// TwinCAT 3 PLC project plc1
// ProgramVersion: 3.1.4024.0
// libraries:
//   SPT Base Types, * (Beckhoff Automation LLC)
//   SPT_XPlanar, * (Beckhoff Automation LLC)
//   Tc2_Standard, * (Beckhoff Automation GmbH)
//   Tc2_System, * (Beckhoff Automation GmbH)
//   Tc3_Mc3PlanarMotion, * (Beckhoff Automation GmbH)
//   Tc3_Module, * (Beckhoff Automation GmbH)
//   Tc3_Physics, * (Beckhoff Automation GmbH)
//   Tc3_XPlanarStandard, * (Beckhoff Automation GmbH)
//   Tc3_XPlanarUtility, * (Beckhoff Automation GmbH & Co. KG)
//   VisuDialogs, * (System)
// project tree:
//   DUTs/ ST_MoverData.TcDUT, ST_StationData.TcDUT
//   / GlobalTextList.TcGTLO, PlcTask.TcTTO, Visualization Manager.TcVMO (not stored)
//   GVLs/ GVL.TcGVL
//   POUs/ FB_ProcessStation.TcPOU, FB_XPlanarModule.TcPOU, MAIN.TcPOU
//   VISUs/ Visualization.TcVIS
//   VISUs/XPlanarObjects/ VisuLayout.TcVIS, VisuMover.TcVIS, VisuStation.TcVIS
// real-time tasks:
//   TASK PlcTask: cycle T#10ms, priority 20, ADS port 350
//   TASK XPlanar Task16: cycle T#250us, priority 1, ADS port 351
//   TASK XPlanar Task17: cycle T#250us, priority 2, ADS port 352
//   TASK MC-Task (MET): cycle T#2ms, priority 3, ADS port 353
//   TASK MC-Task (MPT): cycle T#10ms, priority 4, ADS port 354
//   TASK Job Task: cycle default, priority 5
// variable links:
//   XPlanar MC Project/Axes/Mover4220_1 <-> TcCOM Objects/XPlanar/Mover4220_1
//     IoToMc/STD <-> OutputsToNC3/HWToNC3
//     McToIo/STD <-> InputsFromNC3/NC3ToHW
//   XPlanar MC Project/Axes/Mover4220_2 <-> TcCOM Objects/XPlanar/Mover4220_2
//     McToIo/STD <-> InputsFromNC3/NC3ToHW
//   XPlanar MC Project/Axes/Mover4220_3 <-> TcCOM Objects/XPlanar/Mover4220_3
//     IoToMc/STD <-> OutputsToNC3/HWToNC3
//   TcCOM Objects/XPlanar/Mover4220_2 <-> XPlanar MC Project/Axes/Mover4220_2
//     OutputsToNC3/HWToNC3 <-> IoToMc/STD
//   TcCOM Objects/XPlanar/Mover4220_3 <-> XPlanar MC Project/Axes/Mover4220_3
//     InputsFromNC3/NC3ToHW <-> McToIo/STD
//   plc1 Instance <-> XPlanar MC Project/Axes/Mover4220_1
//     PlcTask Inputs/MAIN.XPlanar1.Movers[1]._Mover.stMoverRef.MCTOPLC/ACT <-> McToPlc/ACT
//     PlcTask Inputs/MAIN.XPlanar1.Movers[1]._Mover.stMoverRef.MCTOPLC/COORDMODE <-> McToPlc/COORDMODE
//     PlcTask Inputs/MAIN.XPlanar1.Movers[1]._Mover.stMoverRef.MCTOPLC/SET <-> McToPlc/SET
//     PlcTask Inputs/MAIN.XPlanar1.Movers[1]._Mover.stMoverRef.MCTOPLC/SETONTRACK <-> McToPlc/SETONTRACK
//     PlcTask Inputs/MAIN.XPlanar1.Movers[1]._Mover.stMoverRef.MCTOPLC/STD <-> McToPlc/STD
//     PlcTask Outputs/MAIN.XPlanar1.Movers[1]._Mover.stMoverRef.PLCTOMC/STD <-> PlcToMc/STD
//   plc1 Instance <-> XPlanar MC Project/Axes/Mover4220_2
//     PlcTask Inputs/MAIN.XPlanar1.Movers[2]._Mover.stMoverRef.MCTOPLC/ACT <-> McToPlc/ACT
//     PlcTask Inputs/MAIN.XPlanar1.Movers[2]._Mover.stMoverRef.MCTOPLC/COORDMODE <-> McToPlc/COORDMODE
//     PlcTask Inputs/MAIN.XPlanar1.Movers[2]._Mover.stMoverRef.MCTOPLC/SET <-> McToPlc/SET
//     PlcTask Inputs/MAIN.XPlanar1.Movers[2]._Mover.stMoverRef.MCTOPLC/SETONTRACK <-> McToPlc/SETONTRACK
//     PlcTask Inputs/MAIN.XPlanar1.Movers[2]._Mover.stMoverRef.MCTOPLC/STD <-> McToPlc/STD
//     PlcTask Outputs/MAIN.XPlanar1.Movers[2]._Mover.stMoverRef.PLCTOMC/STD <-> PlcToMc/STD
//   plc1 Instance <-> XPlanar MC Project/Axes/Mover4220_3
//     PlcTask Inputs/MAIN.XPlanar1.Movers[3]._Mover.stMoverRef.MCTOPLC/ACT <-> McToPlc/ACT
//     PlcTask Inputs/MAIN.XPlanar1.Movers[3]._Mover.stMoverRef.MCTOPLC/COORDMODE <-> McToPlc/COORDMODE
//     PlcTask Inputs/MAIN.XPlanar1.Movers[3]._Mover.stMoverRef.MCTOPLC/SET <-> McToPlc/SET
//     PlcTask Inputs/MAIN.XPlanar1.Movers[3]._Mover.stMoverRef.MCTOPLC/SETONTRACK <-> McToPlc/SETONTRACK
//     PlcTask Inputs/MAIN.XPlanar1.Movers[3]._Mover.stMoverRef.MCTOPLC/STD <-> McToPlc/STD
//     PlcTask Outputs/MAIN.XPlanar1.Movers[3]._Mover.stMoverRef.PLCTOMC/STD <-> PlcToMc/STD
//   plc1 Instance <-> XPlanar MC Project/Groups/Environment
//     PlcTask Inputs/MAIN.XPlanar1.XPlanarTable.XPlanarSystem.environment.MCTOPLC_STD <-> McToPlc/STD
//   plc1 Instance <-> XPlanar MC Project/Groups/Planar Track1
//     PlcTask Inputs/MAIN.XPlanar1.Tracks[1].TrackStandard.stTrackRef.MCTOPLC_STD <-> McToPlc/STD
//   plc1 Instance <-> XPlanar MC Project/Groups/Planar Track2
//     PlcTask Inputs/MAIN.XPlanar1.Tracks[2].TrackStandard.stTrackRef.MCTOPLC_STD <-> McToPlc/STD
//   plc1 Instance <-> XPlanar MC Project/Groups/Planar Track3
//     PlcTask Inputs/MAIN.XPlanar1.Tracks[3].TrackStandard.stTrackRef.MCTOPLC_STD <-> McToPlc/STD
//   plc1 Instance <-> XPlanar MC Project/Groups/XPlanar
//     PlcTask Inputs/MAIN.XPlanar1.XPlanarTable.XPlanarSystem.group.MCTOPLC_STD <-> McToPlc/STD

CONFIGURATION plc1
    RESOURCE PLC ON TwinCAT3
        TASK PlcTask(INTERVAL := T#10ms, PRIORITY := 20);
        PROGRAM MAIN WITH PlcTask : MAIN;
    END_RESOURCE
END_CONFIGURATION

// ---- DUTs/ST_MoverData.TcDUT
TYPE ST_MoverData :
STRUCT
	Status	: int;		// 0- no product, 1- product loaded, 2- product good at station2, 99- product rejected
	PreviousStation	: UDINT;
	DestinationStation	: UDINT;
	
END_STRUCT
END_TYPE

// ---- DUTs/ST_StationData.TcDUT
TYPE ST_StationData :
STRUCT
	Status		: INT;
	VisuPosX 	: INT;
	VisuPosY 	: INT;
//	ProcessTimeAve	: TIME :=T#1S;		// average station process time
//	ProcessTimeAct	: TIME;				// actual (randomized) process time
	
END_STRUCT
END_TYPE

// ---- GVLs/GVL.TcGVL
//{attribute 'qualified_only'}
VAR_GLOBAL

	// mover and station application data
	MoverProcessData 	: ARRAY[1..Tc3_XPlanarStandard.Params_XPlanar.moverCount] OF ST_MoverData;
	StationProcessData 	: ARRAY[1..Tc3_XPlanarStandard.Params_XPlanar.maxNumStation] OF ST_StationData;
	
	iVisuYoffset		: INT := 240;	// vertical offset for visu elements (table Y size)
	CycleCount			: UDINT;

	MoverVelo			: LREAL	:= 400;
	MoverAccel			: LREAL	:= 2000;	
	MoverJerk			: LREAL := 20000;
	MoverGap			: LREAL	:= 200;
	
END_VAR

// ---- POUs/MAIN.TcPOU
PROGRAM MAIN
VAR
	XPlanar1			: FB_XPlanarModule;
	MachineState		: UDINT;
	
	// HMI or PB state triggers
	HmiReset			: BOOL;
	HmiRun				: BOOL;
	HmiStop				: BOOL;	
	HmiDisable			: BOOL;
	
	iNum				: INT;
	
END_VAR

iNum:=iNum+1;

CASE MachineState OF
	0:  // startup
		MachineState := MachineState + 10;

	10:  // wait for Reset / initialize trigger
		IF HmiReset THEN
			HmiReset := FALSE;
			MachineState := MachineState + 10;
		END_IF
		
	20:  // Initialize (assign IPs, build tracks, setup stations, ...)
		IF XPlanar1.Initialize() THEN
			MachineState := MachineState + 10;
		END_IF

	30: // Reset / enable (reset table, enable Group, movers, tracks, ...)
		IF XPlanar1.Reset() THEN
			MachineState := MachineState + 10;
		END_IF
		
	40:  // Recovery (movers join tracks and go to station1)
		XPlanar1.Execute();	// only needed when running or moving movers

		IF XPlanar1.Recovery() THEN
			MachineState := 100;
		END_IF
		
	100:  // Idle, ready to run
		IF HmiRun THEN
			HmiRun := FALSE;
			MachineState := 200;
		END_IF

	200:  // Running
		XPlanar1.Execute();	// only needed when running or moving movers

		IF HmiStop THEN
			HmiStop := FALSE;
			MachineState := 100;
		END_IF
	
	1000:  // Disabled or faulted
		IF HmiReset THEN
			HmiReset := FALSE;
			MachineState := 30;
		END_IF
	
END_CASE

XPlanar1.CyclicLogic();		// top level XPlanar object CyclicLogic method must be called every PLC cycle

// Handle disabling movers
IF (MachineState > 20 AND HmiDisable) 					// monitor disable button after initialized
	OR (MachineState > 90 AND XPlanar1.MoverErr) THEN	// monitor mover error / estop while running
	
	HmiDisable := FALSE;
	XPlanar1.XPlanarTable.XPlanarSystem.DisableMovers();
	MachineState := 1000;
END_IF

END_PROGRAM

// ---- POUs/FB_XPlanarModule.TcPOU
FUNCTION_BLOCK FB_XPlanarModule
VAR_INPUT
END_VAR
VAR_OUTPUT
END_VAR
VAR
	
    XPlanarTable 		: FB_Component_XPlanar 	:= (Name := 'XPlanarTable');
	Station1	 		: FB_ProcessStation		:= (Name := 'Station1');
	Station2	 		: FB_ProcessStation		:= (Name := 'Station2');
	Station3	 		: FB_ProcessStation		:= (Name := 'Station3');

	Movers				: ARRAY[1..Tc3_XPlanarStandard.Params_XPlanar.moverCount] OF FB_XPlanarMover;
	Tracks				: ARRAY[1..Tc3_XPlanarStandard.Params_XPlanar.maxTrackCount] OF FB_XplanarTrackSegment;
	
	MoversTracksInit	: BOOL;	
	MoverErr			: BOOL;
	
END_VAR

// CyclicLogic method must be called every PLC cycle - it calls underlying XPlanar cyclic methods
// Execute method must be called when running or moving movers - manages station state machine
// Initialize method assign Mover and Track IPs, configures and builds tracks & track network, sets up Stations
// Reset method resets objects, enables group, enables movers
// Recovery method sorts movers - join track and go to appropriate station

METHOD CyclicLogic : BOOL
VAR_INPUT
END_VAR
IF NOT MoversTracksInit THEN
	RETURN;
END_IF

XPlanarTable.CyclicLogic();
Station1.CyclicLogic();
Station2.CyclicLogic();
Station3.CyclicLogic();

// Mover error?  (Estopped?)
MoverErr := ip.Movers[1].std.P_ErrorCode<>0 OR ip.Movers[2].std.P_ErrorCode<>0 OR ip.Movers[3].std.P_ErrorCode<>0;
END_METHOD

METHOD Execute : BOOL
VAR_INPUT
END_VAR

VAR
    i 				: UDINT;
END_VAR
// Only needs to be called when running or moving movers for recovery - executes station logic

IF XPlanarTable.InitComplete THEN		
	FOR i := 1 TO Params_XPlanar.maxNumStation DO
		ip.Stations[i].Execute();
	END_FOR
END_IF
END_METHOD

METHOD Initialize : BOOL
VAR_INPUT	
END_VAR

VAR_INST

	i				: UDINT;
	InitState		: UDINT;
	
END_VAR

CASE InitState OF
	
0:
	InitState := InitState + 10;

10: // assign mover and track IPs
	FOR i := 1 TO Tc3_XPlanarStandard.Params_XPlanar.moverCount DO
		Movers[i].MoverIndex := i;
		ip.Movers[i] := Movers[i];
	END_FOR
	
	FOR i := 1 TO Tc3_XPlanarStandard.Params_XPlanar.maxTrackCount DO
		ip.Tracks[i] := Tracks[i];
	END_FOR
	
	MoversTracksInit := TRUE;
	InitState := InitState + 10;
	
20:
	IF XPlanarTable.InitComplete THEN
		InitState := InitState + 10;
	END_IF	

30:  // Set parameters for all tracks - line segments, points, track start/end relationships
	IF SetupTrackSegments() THEN
		InitState := InitState + 10;
	END_IF

40:  // Build and connect all track segments to create track network
	IF XPlanarTable.BuildTracks() THEN
		InitState := InitState + 10;
	END_IF
	
50:  // Set parameters for all stations
	IF SetupStations() THEN
		InitState := InitState + 10;
	END_IF

60:
	Initialize := TRUE;	

END_CASE
END_METHOD

METHOD Recovery : BOOL
VAR_INPUT
END_VAR

VAR_INST
	RecoveryState		: UDINT;
	i					: UDINT;
	JoinTrackNum		: UDINT;
	AllMoversOnTracks	: BOOL;
	GoToStationNum		: UDINT;
	
END_VAR
Recovery := FALSE;

CASE RecoveryState OF
	
0:
	RecoveryState := RecoveryState + 10;

10: // set Mover gap
	FOR i := 1 TO Tc3_XPlanarStandard.Params_XPlanar.moverCount DO
		ip.Movers[i].MoveDynamics.Gap:=MoverGap;	// change default gap
		MoverProcessData[i].Status:=0;	
	END_FOR
	i := 1;
	RecoveryState := 30;

(*  ************* other possible tools / strategies for table recovery ******* 
20: // Dequeue - remove movers from stations
	FOR i := 1 TO Tc3_XPlanarStandard.Params_XPlanar.maxNumStation DO
		ip.Stations[i].MoverQueue.Dequeue();
	END_FOR
	i := 1;
	RecoveryState := 30;
	
	
25: // Station.Recover - get movers back to position within station
	IF ip.Stations[i].Recover() THEN
		i := i + 1;
		IF i > Tc3_XPlanarStandard.Params_XPlanar.maxNumStation THEN
			i := 1;
			RecoveryState := ??;
		END_IF
	END_IF
*)

30: // determine which track to join
	IF ip.Movers[i].std.P_ActPosition.X < 210 THEN
		JoinTrackNum := 1;
	ELSE
		JoinTrackNum := 3;
	END_IF
	
	RecoveryState := RecoveryState + 1;
	
31:	// mover joins track
	IF ip.Movers[i].JoinTrack(ip.Tracks[JoinTrackNum]) THEN
		i := i + 1;
		IF i > Tc3_XPlanarStandard.Params_XPlanar.moverCount THEN
			RecoveryState := RecoveryState + 9;		// all movers handled
		ELSE
			RecoveryState := RecoveryState - 1;		// do next mover
		END_IF
		
	END_IF
	
40:  // verify on track	
	AllMoversOnTracks:=TRUE;
	FOR i := 1 TO Tc3_XPlanarStandard.Params_XPlanar.moverCount DO
//		AllMoversOnTracks := AllMoversOnTracks AND (ip.Movers[i].std.P_TrackId<>0);												// if any mover not on track set False
		AllMoversOnTracks := AllMoversOnTracks AND (ip.Movers[i].std.P_CommandMode = MC_PLANAR_MOVER_COMMAND_MODE.OnTrack);		// if any mover not on track set False
	END_FOR
	
	IF AllMoversOnTracks THEN
		i := 1;
		RecoveryState := RecoveryState + 10;		
	ELSE											// at least on mover not on track
		IF MAIN.HmiDisable THEN
			RecoveryState := 0;						// clear state
		END_IF
	END_IF

50: // determine which station to go to
	IF ip.Movers[i].std.P_ActPosition.Y < 119 THEN
		GoToStationNum := 1;
	ELSIF ip.Movers[i].std.P_ActPosition.X < 210 AND ip.Tracks[3].MoverCount > 1 THEN
		GoToStationNum := 2;
	ELSE
		GoToStationNum := 3;
	END_IF
	
	RecoveryState := RecoveryState + 1;
	
51:	// send movers to stations
	IF ip.Movers[i].SendToStation(ip.Stations[GoToStationNum]) THEN
		i := i + 1;
		IF i > Tc3_XPlanarStandard.Params_XPlanar.moverCount THEN
			RecoveryState := RecoveryState + 9;
		ELSE
			RecoveryState := RecoveryState - 1;		// do next mover
		END_IF
		
	END_IF
	
60:
	Recovery := TRUE;
	RecoveryState := 0;

END_CASE
END_METHOD

METHOD Reset : BOOL
VAR_INPUT
END_VAR

VAR_INST
	ResetState		: UDINT;
	
END_VAR
Reset := FALSE;

CASE ResetState OF
	
0:
	ResetState := 30;

(*	
10:  // Force movers to leave tracks (handles case where movers are still on tracks - support for Recovery method)
	IF XPlanarTable.XPlanarSystem.LeaveTrack() THEN
		ResetState := ResetState + 10;
	END_IF

20:  // Force movers to leave tracks (handles case where movers are still on tracks - support for Recovery method)
	IF XPlanarTable.XPlanarSystem.P_LeaveTrack.Done THEN
		ResetState := ResetState + 10;
	END_IF
*)

30:  // Reset base objects (movers and tracks)
	IF XPlanarTable.Reset() THEN
		ResetState := ResetState + 10;
	END_IF
	
40:  // Enable Group (for CA)
	IF XPlanarTable.EnableGroup() THEN
		ResetState := ResetState + 10;		
	END_IF

50:  // Enable and add movers to Group
	IF XPlanarTable.EnableMovers(UseGroup:=TRUE) THEN
		ResetState := ResetState + 10;		
	END_IF
	
60:  // Enable and add tracks to Group
	IF XPlanarTable.EnableTracks(UseGroup:=TRUE) THEN
		ResetState := ResetState + 10;		
	END_IF	
	
70:
	Reset := TRUE;	
	ResetState := 0;
	
END_CASE
END_METHOD

METHOD PRIVATE SetupStations : BOOL
VAR_INPUT
END_VAR

VAR
	nSta			: UDINT;	// station index
	StationSize 	: UDINT := 50;
END_VAR

nSta := 1;
ip.Stations[nSta] := Station1;							// assign FB to IP
ip.Stations[nSta].ID := nSta;							// set station ID / index
ip.Stations[nSta].TrackID := ip.Tracks[1];				// set rack station is on
ip.Stations[nSta].Position.SetValuesXYC(60, 120, 0);	// station XY location
ip.Stations[nSta].Size.x := StationSize;				// Station size - when station recognizes mover
ip.Stations[nSta].Size.y := StationSize;				
ip.Stations[nSta].StationType := E_StationType.Process;	// (default) process station - Mover stops to 'do' something

GVL.StationProcessData[nSta].VisuPosX:=LREAL_TO_INT(ip.Stations[nSta].Position.x);	// set Visu position
GVL.StationProcessData[nSta].VisuPosY:=LREAL_TO_INT(ip.Stations[nSta].Position.y);

nSta := 2;
ip.Stations[nSta] := Station2;
ip.Stations[nSta].ID := nSta;
ip.Stations[nSta].TrackID := ip.Tracks[2];
ip.Stations[nSta].Position.SetValuesXYC(240, 120, 0);
ip.Stations[nSta].Size.x := StationSize;		
ip.Stations[nSta].Size.y := StationSize;
ip.Stations[nSta].StationType := E_StationType.Process;
ip.Stations[nSta].NextStation := ip.Stations[1];

GVL.StationProcessData[nSta].VisuPosX:=LREAL_TO_INT(ip.Stations[nSta].Position.x);
GVL.StationProcessData[nSta].VisuPosY:=LREAL_TO_INT(ip.Stations[nSta].Position.y);

nSta := 3;
ip.Stations[nSta] := Station3;
ip.Stations[nSta].ID := nSta;
ip.Stations[nSta].TrackID := ip.Tracks[3];
ip.Stations[nSta].Position.SetValuesXYC(420, 120, 0);
ip.Stations[nSta].Size.x := StationSize;
ip.Stations[nSta].Size.y := StationSize;
ip.Stations[nSta].StationType := E_StationType.Process;
ip.Stations[nSta].NextStation := ip.Stations[1];

GVL.StationProcessData[nSta].VisuPosX:=LREAL_TO_INT(ip.Stations[nSta].Position.x);
GVL.StationProcessData[nSta].VisuPosY:=LREAL_TO_INT(ip.Stations[nSta].Position.y);

SetupStations := TRUE;
END_METHOD

METHOD PRIVATE SetupTrackSegments : BOOL
VAR_INST
    nSegmentIndex 		: UDINT;
END_VAR

VAR
    ResultAddPoint 		: INT;

END_VAR
SetupTrackSegments := FALSE;
CASE nSegmentIndex OF
    0: //Get ready
        nSegmentIndex := nSegmentIndex + 1;

    //********************************************************************************************************************************
    //Add states for each track segment in the system
    //********************************************************************************************************************************

    1:
        ip.Tracks[nSegmentIndex].ID := nSegmentIndex;
        IF ip.Tracks[nSegmentIndex].TrackTable.ClearTrackTable() THEN
            ResultAddPoint := ip.Tracks[nSegmentIndex].TrackTable.AddPoint(E_PointType.Line_Start, E_PointOption.none, 	210.0, 60.0, 0.0);
            ResultAddPoint := ip.Tracks[nSegmentIndex].TrackTable.AddPoint(E_PointType.Line_End, E_PointOption.none, 	90.0, 60.0, 0.0);

			ResultAddPoint := ip.Tracks[nSegmentIndex].TrackTable.AddPoint(E_PointType.Line_Start, E_PointOption.none, 	60.0, 90.0, 0.0);
            ResultAddPoint := ip.Tracks[nSegmentIndex].TrackTable.AddPoint(E_PointType.Line_End, E_PointOption.none, 	60.0, 150.0, 0.0);

            ResultAddPoint := ip.Tracks[nSegmentIndex].TrackTable.AddPoint(E_PointType.Line_Start, E_PointOption.none, 	90.0, 180.0, 0.0);
            ResultAddPoint := ip.Tracks[nSegmentIndex].TrackTable.AddPoint(E_PointType.Line_End, E_PointOption.none, 	210.0, 180.0, 0.0);

            ip.Tracks[nSegmentIndex].TrackTable.P_CloseTheLoop := FALSE;
            ip.Tracks[nSegmentIndex].TrackTable.P_StartFromTrack := 0;
            ip.Tracks[nSegmentIndex].TrackTable.P_EndAtTrack     := 0;
			
        END_IF

        nSegmentIndex := nSegmentIndex + 1;

    2:
        ip.Tracks[nSegmentIndex].ID := nSegmentIndex;
        IF ip.Tracks[nSegmentIndex].TrackTable.ClearTrackTable() THEN
            ResultAddPoint := ip.Tracks[nSegmentIndex].TrackTable.AddPoint(E_PointType.Line_Start, E_PointOption.none, 	240.0, 150.0, 0.0);
            ResultAddPoint := ip.Tracks[nSegmentIndex].TrackTable.AddPoint(E_PointType.Line_End, E_PointOption.none, 	240.0, 90.0, 0.0);

            ip.Tracks[nSegmentIndex].TrackTable.P_CloseTheLoop   := FALSE;
            ip.Tracks[nSegmentIndex].TrackTable.P_StartFromTrack := ip.Tracks[1].std;
            ip.Tracks[nSegmentIndex].TrackTable.P_EndAtTrack     := ip.Tracks[1].std;
        END_IF

        nSegmentIndex := nSegmentIndex + 1;

    3:
        ip.Tracks[nSegmentIndex].ID := nSegmentIndex;
        IF ip.Tracks[nSegmentIndex].TrackTable.ClearTrackTable() THEN
            ResultAddPoint := ip.Tracks[nSegmentIndex].TrackTable.AddPoint(E_PointType.Line_Start, E_PointOption.none, 	240.0, 180.0, 0.0);
            ResultAddPoint := ip.Tracks[nSegmentIndex].TrackTable.AddPoint(E_PointType.Line_End, E_PointOption.none, 	390.0, 180.0, 0.0);

            ResultAddPoint := ip.Tracks[nSegmentIndex].TrackTable.AddPoint(E_PointType.Line_Start, E_PointOption.none, 	420.0, 150.0, 0.0);
            ResultAddPoint := ip.Tracks[nSegmentIndex].TrackTable.AddPoint(E_PointType.Line_End, E_PointOption.none, 	420.0, 90.0, 0.0);
			
            ResultAddPoint := ip.Tracks[nSegmentIndex].TrackTable.AddPoint(E_PointType.Line_Start, E_PointOption.none, 	390.0, 60.0, 0.0);
            ResultAddPoint := ip.Tracks[nSegmentIndex].TrackTable.AddPoint(E_PointType.Line_End, E_PointOption.none, 	240.0, 60.0, 0.0);

            ip.Tracks[nSegmentIndex].TrackTable.P_CloseTheLoop   := FALSE;
            ip.Tracks[nSegmentIndex].TrackTable.P_StartFromTrack := ip.Tracks[1].std;
            ip.Tracks[nSegmentIndex].TrackTable.P_EndAtTrack     := ip.Tracks[1].std;
        END_IF

        nSegmentIndex := nSegmentIndex + 1;

    4:
        nSegmentIndex      := 0;
        SetupTrackSegments := TRUE;
END_CASE
END_METHOD

END_FUNCTION_BLOCK

// ---- POUs/FB_ProcessStation.TcPOU
FUNCTION_BLOCK FB_ProcessStation EXTENDS FB_XPlanarStationBase
VAR_INPUT
END_VAR
VAR_OUTPUT
END_VAR
VAR

END_VAR

METHOD Execute

VAR_INST
	ProcessState		: INT;
	tonProcess			: TON;
	Station1Toggle		: BOOL;
	
END_VAR

VAR

END_VAR
SUPER^.Execute();		// executes base station method

IF StationState = E_XPlanarStationState.ProcessMover THEN
		tonProcess(IN:= ProcessState=10, PT:= T#1S, Q=> , ET=> );
	
	CASE ID OF
			
		1:  // Station1 process and decision point
			CASE ProcessState OF
			0:	// init / reset?
				ProcessState := 10;
				
			10: // simulate process with timer
				IF tonProcess.Q THEN ProcessState := 20; END_IF
				
			20:	// after process time, decide what to do next
				GVL.MoverProcessData[ipCurrentMover.MoverIndex].Status := 1;		// product loaded (visu color on)
				IF Station1Toggle THEN
					ipNextStation := ip.Stations[2];
				ELSE
					ipNextStation := ip.Stations[3];
				END_IF
				Station1Toggle := NOT(Station1Toggle);
				CycleCount := CycleCount + 1;
				ProcessState := 100;
			END_CASE

			
		2:  // Station2 process
			CASE ProcessState OF
			0:	// init / reset?
				ProcessState := 10;
				
			10: // simulate process with timer
				IF tonProcess.Q THEN ProcessState := 20; END_IF
				
			20:	// Decide what to do next
				GVL.MoverProcessData[ipCurrentMover.MoverIndex].Status := 0;		// product unloaded (visu off)
				ipNextStation := ip.Stations[1];	
				ProcessState := 100;
			END_CASE			

			
		3:  // Station3 process
			CASE ProcessState OF
			0:	// init / reset?
				ProcessState := 10;
				
			10: // simulate process with timer
				IF tonProcess.Q THEN ProcessState := 20; END_IF
				
			20:	// Decide what to do next
				IF ip.Stations[2].HasMover or ip.Tracks[3].MoverCount > 1 then			// releasing mover to station1 could block mover from getting to Station2
					GVL.MoverProcessData[ipCurrentMover.MoverIndex].Status := 0;		// product unloaded (visu off)
					ipNextStation := ip.Stations[1];	
					ProcessState := 100;
				END_IF
			END_CASE			

			
	END_CASE

	IF ProcessState=100 THEN	// station completed
		// update motion params and gap - could be station specific
		ipCurrentMover.MoveDynamics.Velo := MoverVelo;
		ipCurrentMover.MoveDynamics.Accel := MoverAccel;
		ipCurrentMover.MoveDynamics.Decel := MoverAccel;
		ipCurrentMover.MoveDynamics.Jerk := MoverJerk;
		ipCurrentMover.MoveDynamics.Gap := MoverGap;		
		ProcessState := 0;
		_StationComplete := TRUE;						// process complete - triggers move to next station
	END_IF

END_IF
END_METHOD

END_FUNCTION_BLOCK

// ---- GlobalTextList.TcGTLO
TEXTLIST GlobalTextList
  986 = ' MachineState = %s'
  997 = ' Velocity = %1.1f'
  243 = '%d'
  22 = '%s'
  304 = 'Disable'
  498 = 'Estop'
  409 = 'Initialize'
  454 = 'MachineState = %s'
  687 = 'Reset'
  975 = 'Run'
  55 = 'Start'
  592 = 'Stop'
END_TEXTLIST

// ---- VISUs/Visualization.TcVIS
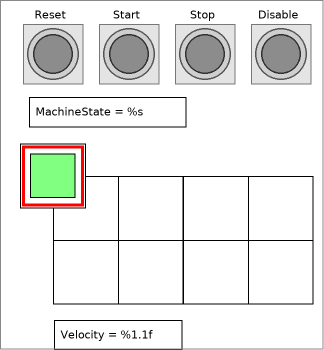
VISUALIZATION Visualization  // 324x350
    Rectangle (29,97 157x30), "MachineState = %s", text variable: MAIN.MachineState
    PushSwitch (23,24 60x60), variable: MAIN.HmiReset, behaviour: TAP, style: Switch-PushSwitch-Gray
    Label (18,5 65x20), "Reset"
    PushSwitch (99,24 60x60), variable: MAIN.HmiRun, behaviour: TAP, style: Switch-PushSwitch-Gray
    Label (94,5 65x20), "Start"
    PushSwitch (175,24 60x60), variable: MAIN.HmiStop, behaviour: TAP, style: Switch-PushSwitch-Gray
    Label (170,5 65x20), "Stop"
    Frame (53,176 271x139)
        shows VisuLayout()
    Rectangle (54,320 128x30), "Velocity = %1.1f", text variable: GVL.MoverVelo
        OnMouseClick: write the text variable via Default, min 5, max 2000
    PushSwitch (251,24 60x60), variable: MAIN.HmiDisable, behaviour: TAP, style: Switch-PushSwitch-Gray
    Label (246,5 65x20), "Disable"
END_VISUALIZATION

// ---- VISUs/XPlanarObjects/VisuLayout.TcVIS
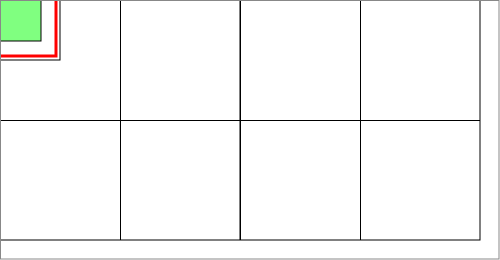
VISUALIZATION VisuLayout  // 500x260
    Group (0,0 240x240)
        Rectangle (0,0 240x240)
        Line (120,0) (120,240)
        Line (0,120) (240,120)
    Group (240,0 240x240)
        Rectangle (0,0 240x240)
        Line (120,0) (120,240)
        Line (0,120) (240,120)
    Frame (-60,-60 120x120)
        shows VisuStation(j := 1)
    Frame (-60,-60 120x120)
        shows VisuStation(j := 2)
    Frame (-60,-60 120x120)
        shows VisuStation(j := 3)
    Frame (-57,-57 114x114)
        shows VisuMover(i := 1)
    Frame (-57,-57 114x114)
        shows VisuMover(i := 2)
    Frame (-57,-57 114x114)
        shows VisuMover(i := 3)
END_VISUALIZATION

// ---- VISUs/XPlanarObjects/VisuMover.TcVIS
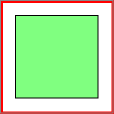
VISUALIZATION VisuMover  // 114x114
VAR_INPUT
	i : INT;
	
END_VAR
    RoundedRectangle (0,0 114x114), "%d", text variable: i
        p3560616238: MAIN.XPlanar1.Movers[i]._Mover.stMoverRef.MCTOPLC.ACT.ActPos.x
        p2738717112: GVL.iVisuYoffset-MAIN.XPlanar1.Movers[i]._Mover.stMoverRef.MCTOPLC.ACT.ActPos.y
        p2858320360: -MAIN.XPlanar1.Movers[i]._Mover.stMoverRef.MCTOPLC.ACT.ActPos.c
    RoundedRectangle (15,15 83x83), colour toggle: GVL.MoverProcessData[i].Status>=99, invisible if: GVL.MoverProcessData[i].Status=0
        p3560616238: MAIN.XPlanar1.Movers[i]._Mover.stMoverRef.MCTOPLC.ACT.ActPos.x
        p2738717112: GVL.iVisuYoffset-MAIN.XPlanar1.Movers[i]._Mover.stMoverRef.MCTOPLC.ACT.ActPos.y
        p2858320360: -MAIN.XPlanar1.Movers[i]._Mover.stMoverRef.MCTOPLC.ACT.ActPos.c
        OnMouseClick: execute { GVL.MoverProcessData[i].Status:=99; }
END_VISUALIZATION

// ---- VISUs/XPlanarObjects/VisuStation.TcVIS
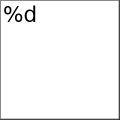
VISUALIZATION VisuStation  // 120x120
VAR_INPUT
	j : INT;
	
END_VAR
    Rectangle (0,0 120x120), "%d", text variable: j
        p3560616238: GVL.StationProcessData[j].VisuPosX
        p2738717112: GVL.iVisuYoffset-GVL.StationProcessData[j].VisuPosY
END_VISUALIZATION
